(* IEC 61131-3 sources: modbus_udp_test/test_2/applications/Core_1_3_2/Защиты, 1 file *)

(* ---- PROTECT.PRG ---- *)
PROGRAM PROTECT
VAR
	protect_control	:	protect_control;
END_VAR

// === IMPLEMENTATION ===

protect_control();

protect_control.SetCommand(MODBUS.SELECTED_PROTECT_OPCUA);

//Показываем состояние выбранной защиты на верхний уровень
IF MODBUS.SELECTED_PROTECT_OPCUA.SelectedNumber <> 0 THEN
	MODBUS.SELECTED_PROTECT_OPCUA.State.DwValue:= MODBUS.PROTECT_STATE[MODBUS.SELECTED_PROTECT_OPCUA.SelectedNumber];
END_IF
